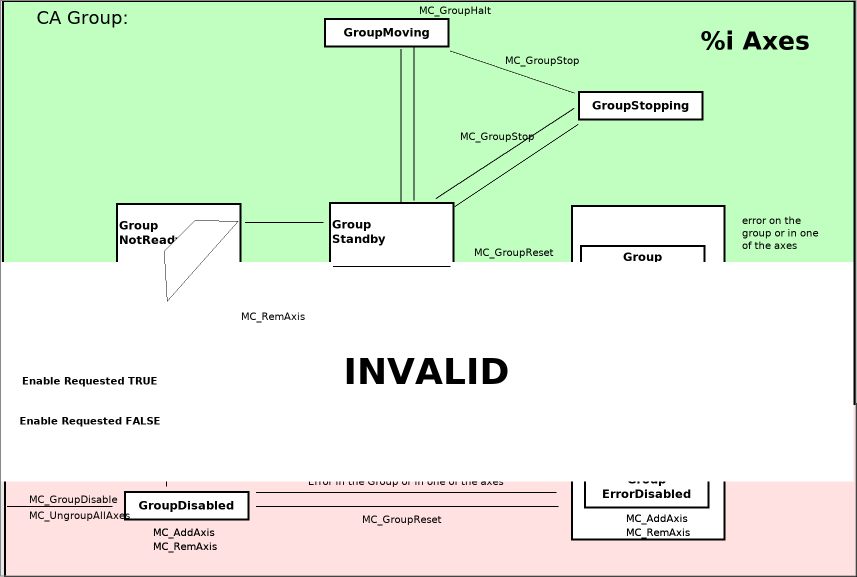
VISUALIZATION FrameAdvancedMotion  // 857x577
VAR_IN_OUT
	stCaGroup			: AXES_GROUP_REF;
END_VAR
    RoundedRectangle (4,403 853x174)
    RoundedRectangle (2,0 853x403)
    RoundedRectangle (324,18 125x29), "GroupMoving", colour toggle: stCaGroup.NcToPlc.Common.GroupStatus.State = 3
    RoundedRectangle (329,202 125x100), "Group Standby", colour toggle: stCaGroup.NcToPlc.Common.GroupStatus.State = 2
    RoundedRectangle (578,91 125x29), "GroupStopping", colour toggle: stCaGroup.NcToPlc.Common.GroupStatus.State = 4
    RoundedRectangle (116,203 125x100), "Group NotReady", colour toggle: stCaGroup.NcToPlc.Common.GroupStatus.State = 7
    RoundedRectangle (571,205 154x335), "GroupErrorStop", colour toggle: stCaGroup.NcToPlc.Common.GroupStatus.State = 5
    RoundedRectangle (124,491 125x29), "GroupDisabled", text variable: stCaGroup.NcToPlc.Common.GroupStatus.State = 1, colour toggle: stCaGroup.NcToPlc.Common.GroupStatus.State = 1
    RoundedRectangle (580,245 125x39), "Group ErrorEnabled"
    RoundedRectangle (584,466 125x42), "Group ErrorDisabled"
    Line (256,506) (558,506)
    Line (167,303) (166,486)
    Line (457,266) (579,266)
    Line (436,198) (574,108)
    Line (414,200) (414,47)
    Group (364,306 62x29)
        Label (0,0 73x15), "MC_AddAxis"
        Label (0,14 74x15), "MC_RemAxis"
    Label (364,306 61x15), "MC_AddAxis"
    Label (364,320 62x15), "MC_RemAxis"
    Group (150,525 62x29)
        Label (0,0 73x15), "MC_AddAxis"
        Label (0,14 74x15), "MC_RemAxis"
    Label (150,525 61x15), "MC_AddAxis"
    Label (150,539 62x15), "MC_RemAxis"
    Group (172,308 62x29)
        Label (0,0 73x15), "MC_AddAxis"
        Label (0,14 74x15), "MC_RemAxis"
    Label (172,308 61x15), "MC_AddAxis"
    Label (172,322 62x15), "MC_RemAxis"
    Group (623,511 62x29)
        Label (0,0 73x15), "MC_AddAxis"
        Label (0,14 74x15), "MC_RemAxis"
    Label (623,511 61x15), "MC_AddAxis"
    Label (623,525 62x15), "MC_RemAxis"
    Group (616,286 62x29)
        Label (0,0 73x15), "MC_AddAxis"
        Label (0,14 74x15), "MC_RemAxis"
    Label (616,286 61x15), "MC_AddAxis"
    Label (616,301 62x15), "MC_RemAxis"
    Label (359,512 77x15), "MC_GroupReset"
    Label (471,245 77x15), "MC_GroupReset"
    Label (26,492 77x15), "MC_GroupDisable"
    Label (416,3 77x15), "MC_GroupHalt"
    Label (502,53 77x15), "MC_GroupStop"
    Label (128,431 77x15), "MC_GroupEnable"
    Line (7,506) (112,506)
    Label (26,508 88x15), "MC_UngroupAllAxes"
    Label (247,272 77x22), "one axis not ready"
    Label (739,215 77x36), "error on the group or in one of the axes"
    Line (401,202) (401,49)
    Line (455,206) (578,124)
    Line (256,492) (556,492)
    Line (245,222) (323,222)
    Label (305,474 170x15), "Error in the Group or in one of the axes"
    Line (233,480) (342,309), "MC_GroupStop"
    Line (234,478) (236,306), "MC_GroupStop"
    Line (246,266) (324,266)
    Line (574,93) (450,51)
    Group (590,294 11x164)
        Line (6,150) (6,0)
        Line (6,161) (13,146)
        Line (5,161) (0,146)
    Line (595,445) (595,293)
    Line (595,457) (600,441)
    Line (594,457) (590,441)
    Group (693,295 11x164)
        Line (6,150) (6,0)
        Line (6,161) (13,146)
        Line (5,161) (0,146)
    Line (698,446) (698,294)
    Line (698,458) (704,442)
    Line (697,458) (693,442)
    Rectangle (0,262 853x219), "INVALID", invisible if: stCaGroup.NcToPlc.Common.GroupStatus.State <> 0
    Label (14,366 152x30), "Enable Requested TRUE", invisible if: stCaGroup.NcToPlc.Common.GroupStatus.Flags.IsEnableRequested = FALSE
    Label (14,406 152x30), "Enable Requested FALSE", invisible if: stCaGroup.NcToPlc.Common.GroupStatus.Flags.IsEnableRequested = TRUE
    Label (457,129 77x15), "MC_GroupStop"
    Polygon (167,301) (164,251) (195,220) (227,221) (238,221)
    Line (333,266) (450,266)
    Label (238,309 60x15), "MC_RemAxis"
    Rectangle (695,10 118x61), "%i Axes", text variable: stCaGroup.NcToPlc.CA.Common.GroupAxesCount
    Rectangle (34,6 97x24), "CA Group:"
END_VISUALIZATION

(* stored: Version 1.1.0.1, ProductVersion 3.1.4024.12
   Visu FrameAdvancedMotion: Id {90e80977-0a75-45b4-9cab-f07c739acc46} *)
